// TwinCAT 3 PLC project Untitled1
// ProgramVersion: 3.1.4022.7
// libraries:
//   Tc2_MC2, * (Beckhoff Automation GmbH)
//   Tc2_Smtp, * (Beckhoff Automation GmbH)
//   Tc2_Standard, * (Beckhoff Automation GmbH)
//   Tc2_System, * (Beckhoff Automation GmbH)
//   Tc3_Module, * (Beckhoff Automation GmbH)
// project tree:
//   DUTs/ ST_Axis.TcDUT (not stored), St_AxisIN.TcDUT (not stored), St_AxisOUT.TcDUT
//   / GlobalTextList.TcGTLO (not stored), PlcTask.TcTTO, Visualization Manager.TcVMO (not stored)
//   GVLs/ GVL_Motion.TcGVL (not stored)
//   POUs/ FB_Motion.TcPOU (not stored), MAIN.TcPOU
// real-time tasks:
//   TASK PlcTask: cycle T#10ms, priority 20, ADS port 350
// motion (NC):
//   TASK NC-Task 1 SAF: cycle T#2ms, priority 4, ADS port 501
//   TASK NC-Task 1 SVB: cycle T#10ms, priority 8, ADS port 511
//   AXIS Axis 1 (id 1)
//     OtherSettings: AllowMotionCmdToSlave=true
//     encoder EncType=8
//       EncPara: MaxCount=#xffffffff
//     drive DrvType=9
//       DrvPara: MaxCount=#xffffffff, DriveControlDWord=#x00030100
//         Analog: ScaleFactorActTorque=0.1
//         TimeComp: TaskDelayCycles=1
//     controller CtrType=1
//       CtrPara: PriorControlFactor=1
//         Observer: BandWidth=20
//   AXIS Axis 2 (id 2)
//     Dynamic: Acceleration=12632, Deceleration=12632, Jerk=37898
//     Velo: RefSearch=84, RefSync=84, SlowManual=421, FastManual=2526, Fast=8421, Maximum=8421
//     OtherSettings: AllowMotionCmdToSlave=true
//     encoder EncType=1
//       EncPara: ScaleFactorNumerator=100, ScaleFactorDenominator=1048576
//     drive DrvType=5
//       Analog: VeloReferenz=9264, ScaleFactorActTorque=0.1
//       TimeComp: TaskDelayCycles=1
//     controller CtrType=1
//       CtrPara: PriorControlFactor=1
//         Observer: BandWidth=20
// I/O:
//   DEVICE Device 1 (EtherCAT) (disabled), AmsNetId 192.168.2.60.2.1
//     Term 1 (EK1200) [EK1200-5000 EtherCAT Power supply (2A E-Bus)]
//       Term 2 (EL1004) [EL1004 4Ch. Dig. Input 24V, 3ms]
//       Term 3 (EL2004) [EL2004 4Ch. Dig. Output 24V, 0.5A]
//       Term 4 (EL3062) [EL3062 2Ch. Ana. Input 0-10V]
//       Term 5 (EL4002) [EL4002 2Ch. Ana. Output 0-10V, 12bit]
//       Term 6 (EK1110) [EK1110 EtherCAT extension]
//     Drive 7 (AX5203-0000-0203) [AX5203-0000-0203 EtherCAT Drive (SoE, 2 Ch.)]
// variable links:
//   NC-Task 1 SAF/Axes/Axis 1 <-> Device 1 (EtherCAT)/Drive 7 (AX5203-0000-0203)
//     Drive/Inputs/In/nDataIn1 <-> AT 1/Following distance
//     Drive/Inputs/In/nDcOutputTime <-> InfoData/DcOutputShift
//     Drive/Inputs/In/nState1 <-> AT 1/Drive status word @bit 8
//     Drive/Inputs/In/nState2 <-> AT 1/Drive status word
//     Drive/Inputs/In/nState4 @bit 1 <-> WcState/InputToggle
//     Drive/Inputs/In/nState4 <-> WcState/WcState
//     Drive/Outputs/Out/nCtrl1 <-> MDT 1/Master control word @bit 8
//     Drive/Outputs/Out/nDataOut1 <-> MDT 1/Position command value
//     Enc/Inputs/In/nDataIn1 <-> AT 1/Position feedback 1 value
//     Enc/Inputs/In/nDcInputTime <-> InfoData/DcInputShift
//     Enc/Inputs/In/nState4 @bit 1 <-> WcState/InputToggle
//     Enc/Inputs/In/nState4 <-> WcState/WcState
//   Untitled1/Untitled1 Instance <-> NC-Task 1 SAF/Axes/Axis 2
//     PlcTask Inputs/GVL_Motion.Axis1.NcToPlc <-> Outputs/ToPlc
//     PlcTask Outputs/GVL_Motion.Axis1.PlcToNc <-> Inputs/FromPlc

CONFIGURATION Untitled1
    RESOURCE PLC ON TwinCAT3
        TASK PlcTask(INTERVAL := T#10ms, PRIORITY := 20);
        PROGRAM MAIN WITH PlcTask : MAIN;
    END_RESOURCE
END_CONFIGURATION

// ---- DUTs/St_AxisOUT.TcDUT
TYPE St_AxisOUT :
STRUCT
	
bPowerErr	:	BOOL;
bPowerBusy	:	BOOL;
bPowerActive	:	BOOL;
bPowerStat	:	BOOL;
bPowErrid	:	UDINT;

bAbsErr		:	BOOL;
bAbsActive	:	BOOL;
bAbsBusy	:	BOOL;
bAbsDone	:	BOOL;

bStopErr	:	BOOL;
bStopBusy	:	BOOL;
bStopActive	:	BOOL;
bStopDone	:	BOOL;

bResetErr	:	BOOL;
bResetBusy	:	BOOL;
bResetDone	:	BOOL;

END_STRUCT
END_TYPE

// ---- POUs/MAIN.TcPOU
PROGRAM MAIN
VAR
		
	nState: INT;
	sMsg	:	STRING :=	'Sistemde Hata Olustu	Hata Kodu	=	 ';
	sMsg2	: 	STRING;
	sVar	:	STRING;
		
	bSend	:	BOOL;
	bErr	:	BOOL;
	bBusy	:	BOOL;
	bExecute: BOOL;
	
	sAxis	:	ST_Axis;
	fbmail: FB_SmtpV3;
	fbMotion: FB_Motion;

	sMsg3: STRING;
	sVar2: STRING(255);
	F_TRIG1: F_TRIG;
	Sens1: BOOL;
	counter: INT;
END_VAR


fbMotion(Axis:= .Axis1 , StAxis:=sAxis);
ACT_System();

ACTION ACT_System:

	fbmail(
	sNetId:='192.168.48.1.1.1' , 
	sSmtpServer:='smtp.gmail.com' , 
	sUsername:= '*******@gmail.com', 
	sPassword:= '*********',         
	nEncryption:= 2,                 
	sFrom:= '********@gmail.com',    
	sTo:= '**********@gmail.com',    
	sCc:= , 
	sBcc:= , 
	sSubject:= 'Sistem Hatasi Mevcut', 
	pMessage:= , 
	cbMessage:= , 
	bExecute:=bSend , 
	tTimeout:=T#2S , 
	bBusy=>bBusy , 
	bError=>bErr , 
	nErrId=> );

	F_TRIG1(CLK:=Sens1 , Q=> );

	

	sMsg2	:=	UDINT_TO_STRING(axis2.NcToPlc.ErrorCode);
	sMsg3	:=	UDINT_TO_STRING(saxis.OUTPUT.bPowErrid);
	
	sVar	:=	CONCAT(STR1:=sMsg , STR2:=sMsg2 );
	sVar2	:=	CONCAT(STR1:=sMsg , STR2:=sMsg3 );
	
	sAxis.INPUT.fOverride	:=	100;
	sAxis.INPUT.bStop	:= FALSE;
	
CASE nState OF
	
	0:
	
		saxis.INPUT.bMoveAbs	:=	FALSE;

		IF  saxis.OUTPUT.bPowerActive
		AND NOT sAxis.OUTPUT.bAbsErr	
		AND saxis.OUTPUT.bPowerActive
		AND sAxis.OUTPUT.bPowerStat THEN
		 
			nState	:=	1;
						
		END_IF
		
	1:
				
		IF bExecute 
		AND NOT sAxis.OUTPUT.bPowerErr
		AND sAxis.OUTPUT.bPowerActive 
		AND NOT sAxis.OUTPUT.bStopActive THEN
		
			nState	:=	10;
		
		ELSIF sAxis.OUTPUT.bAbsErr THEN
			nState:=999;
		END_IF
		
	10:			
		sAxis.INPUT.bStop	:=	FALSE;
		sAxis.INPUT.bMoveAbs	:=	TRUE;
		sAxis.INPUT.fPosition	:= 10000;
		sAxis.INPUT.nVelocity	:=	5000;
		
		IF	sAxis.OUTPUT.bAbsBusy 
		AND NOT sAxis.OUTPUT.bPowerErr
		AND sAxis.OUTPUT.bPowerActive 
		AND NOT sAxis.OUTPUT.bStopActive THEN
					
			nState	:=	20;
				
		ELSIF sAxis.OUTPUT.bAbsErr THEN
			nState:=999;
		END_IF

	20:

		IF sAxis.OUTPUT.bAbsDone 
		AND NOT sAxis.OUTPUT.bPowerErr	
		AND NOT sAxis.OUTPUT.bAbsErr	
		AND saxis.OUTPUT.bPowerActive	THEN

			nState	:=	30;
			sAxis.INPUT.bMoveAbs	:=	FALSE;
				
		ELSIF sAxis.OUTPUT.bAbsErr THEN
			nState:=999;
		END_IF
			
	30:	
		sAxis.INPUT.bStop	:=	FALSE;
		sAxis.INPUT.bMoveAbs	:=	TRUE;
		sAxis.INPUT.fPosition	:= 45000;
		sAxis.INPUT.nVelocity	:=	7000;
			
		
		
			IF	sAxis.OUTPUT.bAbsBusy 
			AND NOT sAxis.OUTPUT.bPowerErr
			AND sAxis.OUTPUT.bPowerActive 
			AND NOT sAxis.OUTPUT.bStopActive THEN							
				nState	:=	40;		
			ELSIF sAxis.OUTPUT.bAbsErr THEN
				nState:=999;
			END_IF
	
				
	40:
		IF sAxis.OUTPUT.bAbsDone 
		AND NOT sAxis.OUTPUT.bPowerErr	
		AND NOT sAxis.OUTPUT.bAbsErr	
		AND saxis.OUTPUT.bPowerActive	THEN

		
			sAxis.INPUT.bMoveAbs	:=	FALSE;

			IF f_trig1.Q THEN
					
				counter	:=	counter	+	1;

				IF counter >=5 THEN
					counter	:=	0;
					nState	:=	50;
				END_IF
			
			END_IF

			
				
			ELSIF sAxis.OUTPUT.bAbsErr THEN
				nState:=999;
			END_IF
					
				
		50:	
			sAxis.INPUT.bStop	:=	FALSE;
			sAxis.INPUT.bMoveAbs	:=	TRUE;
			sAxis.INPUT.fPosition	:= 0;
			sAxis.INPUT.nVelocity	:=	7000;
		
			IF	sAxis.OUTPUT.bAbsBusy AND NOT	sAxis.OUTPUT.bPowerErr	
			AND NOT	sAxis.OUTPUT.bAbsErr	THEN
					
				nState	:=	60;
				
			ELSIF sAxis.OUTPUT.bAbsErr THEN
				nState:=999;
			END_IF
			
		60:

			IF sAxis.OUTPUT.bAbsDone AND NOT sAxis.OUTPUT.bPowerErr	
			AND NOT	sAxis.OUTPUT.bAbsErr	THEN

				nState	:=	0;
				sAxis.INPUT.bMoveAbs	:=	FALSE;
				
			ELSIF sAxis.OUTPUT.bAbsErr THEN
				nState:=999;
			END_IF
				
		999:
		
    	
			// Hataya neden olacak hata kodunu atacak şekilde düzenle
		
			saxis.INPUT.bReset	:=	TRUE;
			saxis.INPUT.bMoveAbs	:=	FALSE;
			
			fbmail.pMessage	:=	ADR(sVAr);
			fbmail.cbMessage	:=	SIZEOF(sVar);
			bSend	:=	TRUE;	
    		
		
			IF saxis.OUTPUT.bResetDone THEN
				nState	:=	1000;
			END_IF
			
		1000:
			
			IF NOT sAxis.OUTPUT.bPowerErr 
			AND NOT saxis.OUTPUT.bAbsErr
			AND saxis.OUTPUT.bPowerActive
			AND NOT saxis.OUTPUT.bPowerErr THEN
				
				bSend	:=	FALSE;
				nState	:=	0;
			
			END_IF
        	
	
END_CASE


	IF NOT bExecute THEN
		nState	:=	0;
		
		sAxis.INPUT.bStop	:=	TRUE;
		saxis.INPUT.bMoveAbs	:=	FALSE;
		
		sAxis.INPUT.fPosition	:= 0;
		sAxis.INPUT.nVelocity	:=	0;

			IF saxis.OUTPUT.bStopDone AND NOT sAxis.OUTPUT.bPowerErr 
			AND sAxis.OUTPUT.bPowerActive THEN
					sAxis.INPUT.bStop	:=	FALSE;
					nState	:=	0;
			END_IF
	END_IF

			
	
		IF 	saxis.OUTPUT.bPowerErr THEN
	
			fbmail.pMessage	:=	ADR(sVAr2);
			fbmail.cbMessage	:=	SIZEOF(sVar2);
			bSend	:=	TRUE;
		
			saxis.INPUT.bReset	:=	TRUE;
			
				IF saxis.OUTPUT.bResetDone 
				AND NOT saxis.OUTPUT.bAbsErr 
				AND NOT saxis.OUTPUT.bPowerErr THEN
					
					bSend	:=	FALSE;
					saxis.INPUT.bMoveAbs	:=	FALSE;
					nState	:=	0;
				
				END_IF
			END_IF
END_ACTION

END_PROGRAM
